(* PLC project AW9523B, INSA Strasbourg AW9523B 1.0, author Mathieu Giamberini *)
(* stored: creationDateTime 2024-11-13T08:40:00, modificationDateTime 2024-10-04T15:56:57 *)

TYPE AW9523B : STRUCT
  Address : BYTE := 16#00;
  Init : BOOL := False;
  P1 : BYTE := 2#00000000;
  P2 : BYTE := 2#00000000;
END_STRUCT;
END_TYPE

(* Return the state of the specified pin on the specified AW9523B board *)
FUNCTION_BLOCK DI_1
  VAR_INPUT
    B_AD : BYTE;  (* Board I2C Address *)
    P_AD : BYTE;  (* Pin Address *)
  END_VAR
  VAR_OUTPUT
    PIN : BOOL;  (* Pin state *)
  END_VAR

            
          
END_FUNCTION_BLOCK

(* Set the state of the specified pin on the specified AW9523B board *)
FUNCTION_BLOCK DQ_1
  VAR_INPUT
    B_AD : BYTE;  (* Board I2C Address *)
    P_AD : BYTE;  (* Pin Address *)
    PIN : BOOL;  (* Pin state *)
  END_VAR

            
          
END_FUNCTION_BLOCK

(* Return the states of the specified pins on the specified AW9523B board *)
FUNCTION_BLOCK DI_8
  VAR_INPUT
    B_AD : BYTE;  (* Board I2C Address *)
    X : BOOL;  (* Pins side *)
  END_VAR
  VAR_OUTPUT
    PX_0 : BOOL;  (* Pin x_0 state *)
    PX_1 : BOOL;  (* Pin x_1 state *)
    PX_2 : BOOL;  (* Pin x_2 state *)
    PX_3 : BOOL;  (* Pin x_3 state *)
    PX_4 : BOOL;  (* Pin x_4 state *)
    PX_5 : BOOL;  (* Pin x_5 state *)
    PX_6 : BOOL;  (* Pin x_6 state *)
    PX_7 : BOOL;  (* Pin x_7 state *)
  END_VAR

            
          
END_FUNCTION_BLOCK

(* Set the states of the specified pins on the specified AW9523B board *)
FUNCTION_BLOCK DQ_8
  VAR_INPUT
    B_AD : BYTE;  (* Board I2C Address *)
    X : BOOL;  (* Pins side *)
    PX_0 : BOOL;  (* Pin x_0 state *)
    PX_1 : BOOL;  (* Pin x_1 state *)
    PX_2 : BOOL;  (* Pin x_2 state *)
    PX_3 : BOOL;  (* Pin x_3 state *)
    PX_4 : BOOL;  (* Pin x_4 state *)
    PX_5 : BOOL;  (* Pin x_5 state *)
    PX_6 : BOOL;  (* Pin x_6 state *)
    PX_7 : BOOL;  (* Pin x_7 state *)
  END_VAR

            
          
END_FUNCTION_BLOCK
